(* Logix 5000 project; controller AMANA_DC_PLANT_01 vendor 1 type 14 code 164 rev 31.12; software revision 31.02; part 7 of 9 *)
(* tags used below, declared in another part *)
   Barcode_Longest : DINT;
   Barcode_Shortest : DINT;
   Comma : STRING;
   Counters : COUNTER[16];
   NULL_String : STRING;
   PRE_SET_COMMA_POSITION_1 : DINT;
   SCANNER_ClearPack_DATA : Keyence_2_Barcode;
   SCANNER_LN4_DATA : Keyence_2_Barcode;
   SCANNER_LN67MERGE_DATA : Keyence_2_Barcode;
   SCANNER_LN6_DATA : Keyence_2_Barcode;
   SCANNER_LN7_DATA : Keyence_2_Barcode;
   Read_From_Clearpack : INT[16];
(* OH_BARCODE_SCAN, continued *)

ROUTINE R01_CLEARPACK   (* ladder *)
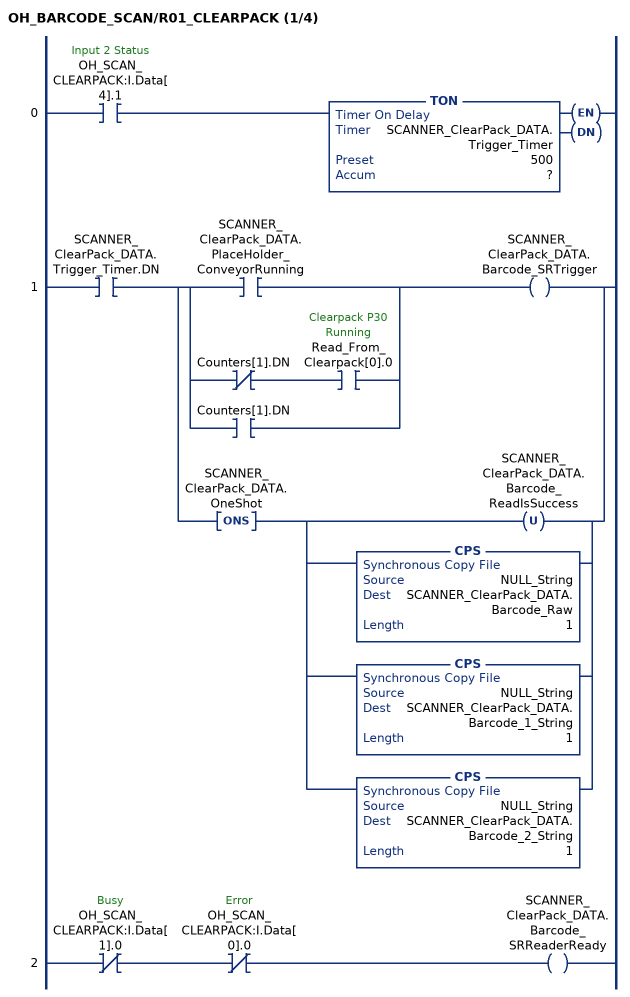
   0: XIC(OH_SCAN_CLEARPACK:I.Data[4].1)TON(SCANNER_ClearPack_DATA.Trigger_Timer,?,?);
   1: XIC(SCANNER_ClearPack_DATA.Trigger_Timer.DN)[[XIC(SCANNER_ClearPack_DATA.PlaceHolder_ConveyorRunning) ,XIO(Counters[1].DN) XIC(Read_From_Clearpack[0].0) ,XIC(Counters[1].DN) ] OTE(SCANNER_ClearPack_DATA.Barcode_SRTrigger) ,ONS(SCANNER_ClearPack_DATA.OneShot) [OTU(SCANNER_ClearPack_DATA.Barcode_ReadIsSuccess) ,CPS(NULL_String,SCANNER_ClearPack_DATA.Barcode_Raw,1) ,CPS(NULL_String,SCANNER_ClearPack_DATA.Barcode_1_String,1) ,CPS(NULL_String,SCANNER_ClearPack_DATA.Barcode_2_String,1) ] ];
   2: XIO(OH_SCAN_CLEARPACK:I.Data[1].0)XIO(OH_SCAN_CLEARPACK:I.Data[0].0)OTE(SCANNER_ClearPack_DATA.Barcode_SRReaderReady);
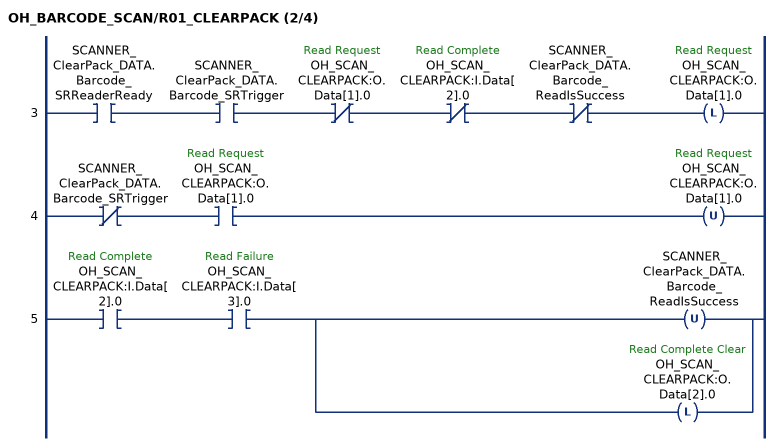
   3: XIC(SCANNER_ClearPack_DATA.Barcode_SRReaderReady)XIC(SCANNER_ClearPack_DATA.Barcode_SRTrigger)XIO(OH_SCAN_CLEARPACK:O.Data[1].0)XIO(OH_SCAN_CLEARPACK:I.Data[2].0)XIO(SCANNER_ClearPack_DATA.Barcode_ReadIsSuccess)OTL(OH_SCAN_CLEARPACK:O.Data[1].0);
   4: XIO(SCANNER_ClearPack_DATA.Barcode_SRTrigger)XIC(OH_SCAN_CLEARPACK:O.Data[1].0)OTU(OH_SCAN_CLEARPACK:O.Data[1].0);
   5: XIC(OH_SCAN_CLEARPACK:I.Data[2].0)XIC(OH_SCAN_CLEARPACK:I.Data[3].0)[OTU(SCANNER_ClearPack_DATA.Barcode_ReadIsSuccess) ,OTL(OH_SCAN_CLEARPACK:O.Data[2].0) ];
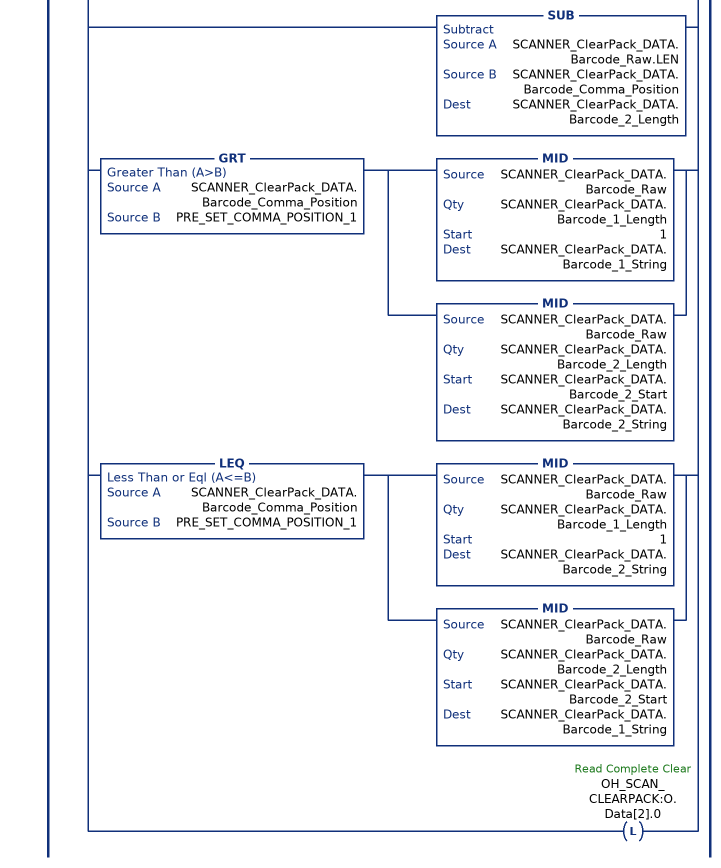
   6: XIC(OH_SCAN_CLEARPACK:I.Data[2].0)XIO(OH_SCAN_CLEARPACK:I.Data[3].0)LIM(Barcode_Shortest,OH_SCAN_CLEARPACK:I.Data[42],Barcode_Longest)[OTL(SCANNER_ClearPack_DATA.Barcode_ReadIsSuccess) ,SUB(OH_SCAN_CLEARPACK:I.Data[42],1,SCANNER_ClearPack_DATA.Barcode_Raw.LEN) ,CPS(OH_SCAN_CLEARPACK:I.Data[44],SCANNER_ClearPack_DATA.Barcode_Raw.DATA[0],SCANNER_ClearPack_DATA.Barcode_Raw.LEN) ,FIND(SCANNER_ClearPack_DATA.Barcode_Raw,Comma,1,SCANNER_ClearPack_DATA.Barcode_Comma_Position) ,SUB(SCANNER_ClearPack_DATA.Barcode_Comma_Position,1,SCANNER_ClearPack_DATA.Barcode_1_Length) ,ADD(SCANNER_ClearPack_DATA.Barcode_Comma_Position,1,SCANNER_ClearPack_DATA.Barcode_2_Start) ,SUB(SCANNER_ClearPack_DATA.Barcode_Raw.LEN,SCANNER_ClearPack_DATA.Barcode_Comma_Position,SCANNER_ClearPack_DATA.Barcode_2_Length) ,GRT(SCANNER_ClearPack_DATA.Barcode_Comma_Position,PRE_SET_COMMA_POSITION_1) [MID(SCANNER_ClearPack_DATA.Barcode_Raw,SCANNER_ClearPack_DATA.Barcode_1_Length,1,SCANNER_ClearPack_DATA.Barcode_1_String) ,MID(SCANNER_ClearPack_DATA.Barcode_Raw,SCANNER_ClearPack_DATA.Barcode_2_Length,SCANNER_ClearPack_DATA.Barcode_2_Start,SCANNER_ClearPack_DATA.Barcode_2_String) ] ,LEQ(SCANNER_ClearPack_DATA.Barcode_Comma_Position,PRE_SET_COMMA_POSITION_1) [MID(SCANNER_ClearPack_DATA.Barcode_Raw,SCANNER_ClearPack_DATA.Barcode_1_Length,1,SCANNER_ClearPack_DATA.Barcode_2_String) ,MID(SCANNER_ClearPack_DATA.Barcode_Raw,SCANNER_ClearPack_DATA.Barcode_2_Length,SCANNER_ClearPack_DATA.Barcode_2_Start,SCANNER_ClearPack_DATA.Barcode_1_String) ] ,OTL(OH_SCAN_CLEARPACK:O.Data[2].0) ];
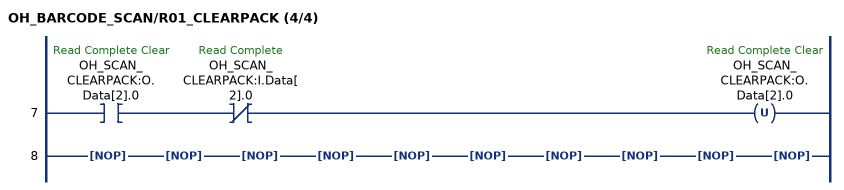
   7: XIC(OH_SCAN_CLEARPACK:O.Data[2].0)XIO(OH_SCAN_CLEARPACK:I.Data[2].0)OTU(OH_SCAN_CLEARPACK:O.Data[2].0);
   8: NOP()NOP()NOP()NOP()NOP()NOP()NOP()NOP()NOP()NOP();
END_ROUTINE

ROUTINE R02_LN4   (* ladder *)
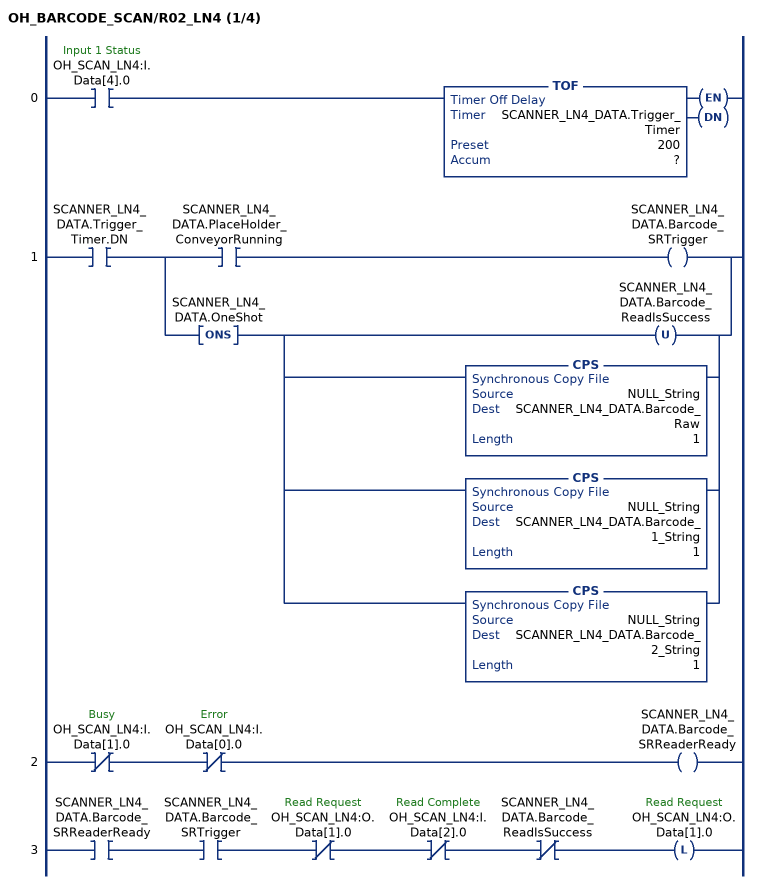
   0: XIC(OH_SCAN_LN4:I.Data[4].0)TOF(SCANNER_LN4_DATA.Trigger_Timer,?,?);
   1: XIC(SCANNER_LN4_DATA.Trigger_Timer.DN)[XIC(SCANNER_LN4_DATA.PlaceHolder_ConveyorRunning) OTE(SCANNER_LN4_DATA.Barcode_SRTrigger) ,ONS(SCANNER_LN4_DATA.OneShot) [OTU(SCANNER_LN4_DATA.Barcode_ReadIsSuccess) ,CPS(NULL_String,SCANNER_LN4_DATA.Barcode_Raw,1) ,CPS(NULL_String,SCANNER_LN4_DATA.Barcode_1_String,1) ,CPS(NULL_String,SCANNER_LN4_DATA.Barcode_2_String,1) ] ];
   2: XIO(OH_SCAN_LN4:I.Data[1].0)XIO(OH_SCAN_LN4:I.Data[0].0)OTE(SCANNER_LN4_DATA.Barcode_SRReaderReady);
   3: XIC(SCANNER_LN4_DATA.Barcode_SRReaderReady)XIC(SCANNER_LN4_DATA.Barcode_SRTrigger)XIO(OH_SCAN_LN4:O.Data[1].0)XIO(OH_SCAN_LN4:I.Data[2].0)XIO(SCANNER_LN4_DATA.Barcode_ReadIsSuccess)OTL(OH_SCAN_LN4:O.Data[1].0);
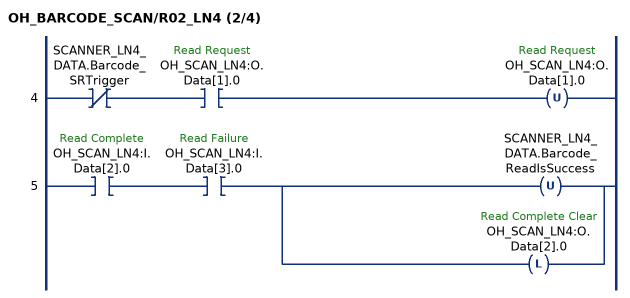
   4: XIO(SCANNER_LN4_DATA.Barcode_SRTrigger)XIC(OH_SCAN_LN4:O.Data[1].0)OTU(OH_SCAN_LN4:O.Data[1].0);
   5: XIC(OH_SCAN_LN4:I.Data[2].0)XIC(OH_SCAN_LN4:I.Data[3].0)[OTU(SCANNER_LN4_DATA.Barcode_ReadIsSuccess) ,OTL(OH_SCAN_LN4:O.Data[2].0) ];
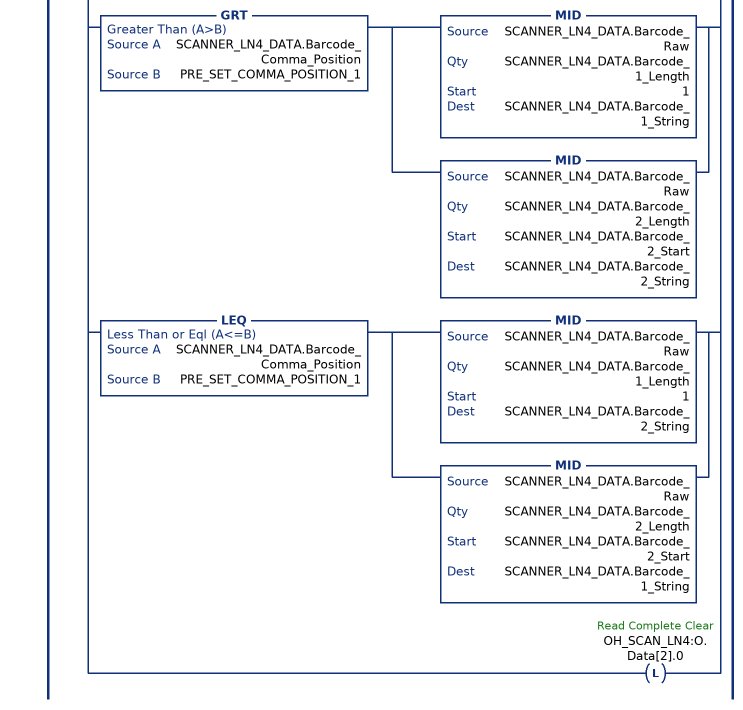
   6: XIC(OH_SCAN_LN4:I.Data[2].0)XIO(OH_SCAN_LN4:I.Data[3].0)LIM(Barcode_Shortest,OH_SCAN_LN4:I.Data[42],Barcode_Longest)[OTL(SCANNER_LN4_DATA.Barcode_ReadIsSuccess) ,SUB(OH_SCAN_LN4:I.Data[42],1,SCANNER_LN4_DATA.Barcode_Raw.LEN) ,CPS(OH_SCAN_LN4:I.Data[44],SCANNER_LN4_DATA.Barcode_Raw.DATA[0],SCANNER_LN4_DATA.Barcode_Raw.LEN) ,FIND(SCANNER_LN4_DATA.Barcode_Raw,Comma,1,SCANNER_LN4_DATA.Barcode_Comma_Position) ,SUB(SCANNER_LN4_DATA.Barcode_Comma_Position,1,SCANNER_LN4_DATA.Barcode_1_Length) ,ADD(SCANNER_LN4_DATA.Barcode_Comma_Position,1,SCANNER_LN4_DATA.Barcode_2_Start) ,SUB(SCANNER_LN4_DATA.Barcode_Raw.LEN,SCANNER_LN4_DATA.Barcode_Comma_Position,SCANNER_LN4_DATA.Barcode_2_Length) ,GRT(SCANNER_LN4_DATA.Barcode_Comma_Position,PRE_SET_COMMA_POSITION_1) [MID(SCANNER_LN4_DATA.Barcode_Raw,SCANNER_LN4_DATA.Barcode_1_Length,1,SCANNER_LN4_DATA.Barcode_1_String) ,MID(SCANNER_LN4_DATA.Barcode_Raw,SCANNER_LN4_DATA.Barcode_2_Length,SCANNER_LN4_DATA.Barcode_2_Start,SCANNER_LN4_DATA.Barcode_2_String) ] ,LEQ(SCANNER_LN4_DATA.Barcode_Comma_Position,PRE_SET_COMMA_POSITION_1) [MID(SCANNER_LN4_DATA.Barcode_Raw,SCANNER_LN4_DATA.Barcode_1_Length,1,SCANNER_LN4_DATA.Barcode_2_String) ,MID(SCANNER_LN4_DATA.Barcode_Raw,SCANNER_LN4_DATA.Barcode_2_Length,SCANNER_LN4_DATA.Barcode_2_Start,SCANNER_LN4_DATA.Barcode_1_String) ] ,OTL(OH_SCAN_LN4:O.Data[2].0) ];
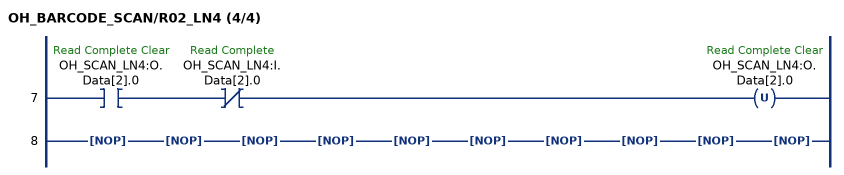
   7: XIC(OH_SCAN_LN4:O.Data[2].0)XIO(OH_SCAN_LN4:I.Data[2].0)OTU(OH_SCAN_LN4:O.Data[2].0);
   8: NOP()NOP()NOP()NOP()NOP()NOP()NOP()NOP()NOP()NOP();
END_ROUTINE

ROUTINE R03_LN6   (* ladder *)
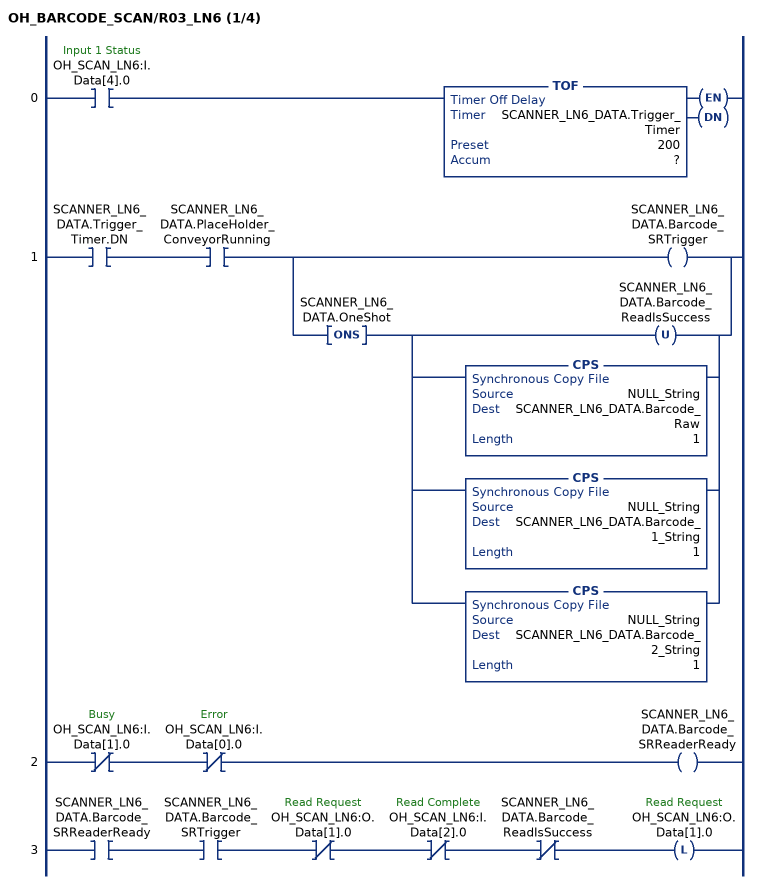
   0: XIC(OH_SCAN_LN6:I.Data[4].0)TOF(SCANNER_LN6_DATA.Trigger_Timer,?,?);
   1: XIC(SCANNER_LN6_DATA.Trigger_Timer.DN)XIC(SCANNER_LN6_DATA.PlaceHolder_ConveyorRunning)[OTE(SCANNER_LN6_DATA.Barcode_SRTrigger) ,ONS(SCANNER_LN6_DATA.OneShot) [OTU(SCANNER_LN6_DATA.Barcode_ReadIsSuccess) ,CPS(NULL_String,SCANNER_LN6_DATA.Barcode_Raw,1) ,CPS(NULL_String,SCANNER_LN6_DATA.Barcode_1_String,1) ,CPS(NULL_String,SCANNER_LN6_DATA.Barcode_2_String,1) ] ];
   2: XIO(OH_SCAN_LN6:I.Data[1].0)XIO(OH_SCAN_LN6:I.Data[0].0)OTE(SCANNER_LN6_DATA.Barcode_SRReaderReady);
   3: XIC(SCANNER_LN6_DATA.Barcode_SRReaderReady)XIC(SCANNER_LN6_DATA.Barcode_SRTrigger)XIO(OH_SCAN_LN6:O.Data[1].0)XIO(OH_SCAN_LN6:I.Data[2].0)XIO(SCANNER_LN6_DATA.Barcode_ReadIsSuccess)OTL(OH_SCAN_LN6:O.Data[1].0);
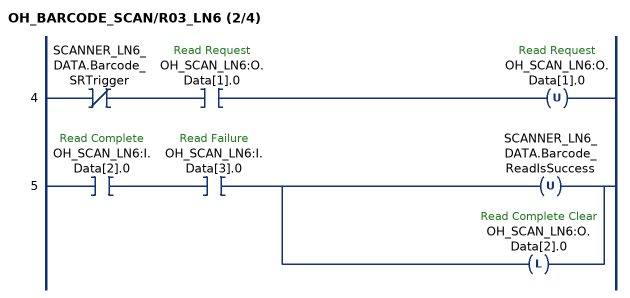
   4: XIO(SCANNER_LN6_DATA.Barcode_SRTrigger)XIC(OH_SCAN_LN6:O.Data[1].0)OTU(OH_SCAN_LN6:O.Data[1].0);
   5: XIC(OH_SCAN_LN6:I.Data[2].0)XIC(OH_SCAN_LN6:I.Data[3].0)[OTU(SCANNER_LN6_DATA.Barcode_ReadIsSuccess) ,OTL(OH_SCAN_LN6:O.Data[2].0) ];
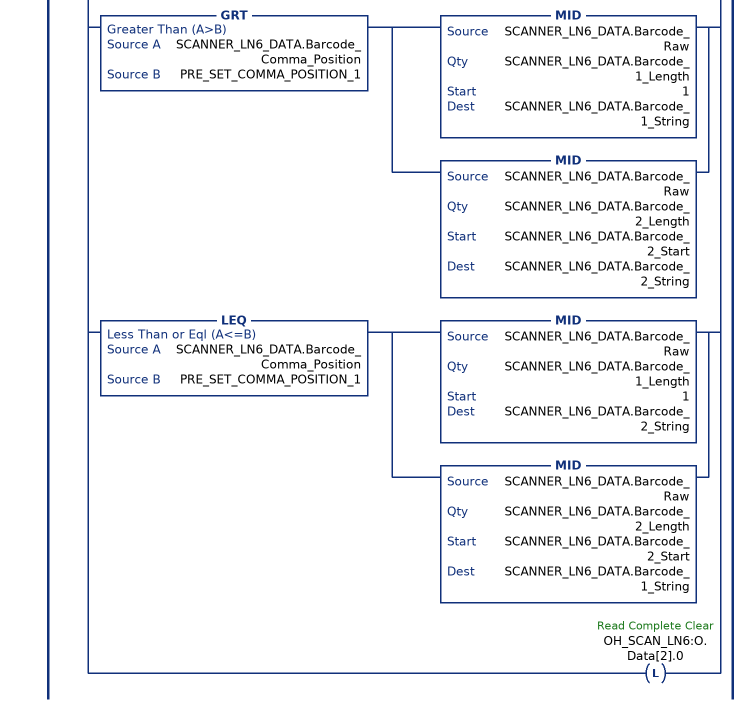
   6: XIC(OH_SCAN_LN6:I.Data[2].0)XIO(OH_SCAN_LN6:I.Data[3].0)LIM(Barcode_Shortest,OH_SCAN_LN6:I.Data[42],Barcode_Longest)[OTL(SCANNER_LN6_DATA.Barcode_ReadIsSuccess) ,SUB(OH_SCAN_LN6:I.Data[42],1,SCANNER_LN6_DATA.Barcode_Raw.LEN) ,CPS(OH_SCAN_LN6:I.Data[44],SCANNER_LN6_DATA.Barcode_Raw.DATA[0],SCANNER_LN6_DATA.Barcode_Raw.LEN) ,FIND(SCANNER_LN6_DATA.Barcode_Raw,Comma,1,SCANNER_LN6_DATA.Barcode_Comma_Position) ,SUB(SCANNER_LN6_DATA.Barcode_Comma_Position,1,SCANNER_LN6_DATA.Barcode_1_Length) ,ADD(SCANNER_LN6_DATA.Barcode_Comma_Position,1,SCANNER_LN6_DATA.Barcode_2_Start) ,SUB(SCANNER_LN6_DATA.Barcode_Raw.LEN,SCANNER_LN6_DATA.Barcode_Comma_Position,SCANNER_LN6_DATA.Barcode_2_Length) ,GRT(SCANNER_LN6_DATA.Barcode_Comma_Position,PRE_SET_COMMA_POSITION_1) [MID(SCANNER_LN6_DATA.Barcode_Raw,SCANNER_LN6_DATA.Barcode_1_Length,1,SCANNER_LN6_DATA.Barcode_1_String) ,MID(SCANNER_LN6_DATA.Barcode_Raw,SCANNER_LN6_DATA.Barcode_2_Length,SCANNER_LN6_DATA.Barcode_2_Start,SCANNER_LN6_DATA.Barcode_2_String) ] ,LEQ(SCANNER_LN6_DATA.Barcode_Comma_Position,PRE_SET_COMMA_POSITION_1) [MID(SCANNER_LN6_DATA.Barcode_Raw,SCANNER_LN6_DATA.Barcode_1_Length,1,SCANNER_LN6_DATA.Barcode_2_String) ,MID(SCANNER_LN6_DATA.Barcode_Raw,SCANNER_LN6_DATA.Barcode_2_Length,SCANNER_LN6_DATA.Barcode_2_Start,SCANNER_LN6_DATA.Barcode_1_String) ] ,OTL(OH_SCAN_LN6:O.Data[2].0) ];
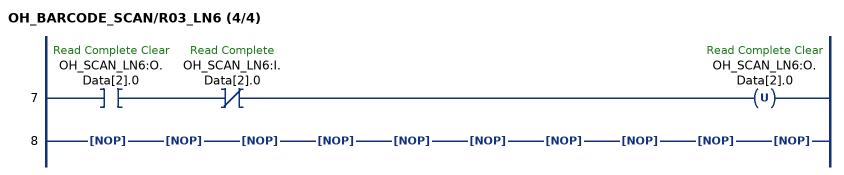
   7: XIC(OH_SCAN_LN6:O.Data[2].0)XIO(OH_SCAN_LN6:I.Data[2].0)OTU(OH_SCAN_LN6:O.Data[2].0);
   8: NOP()NOP()NOP()NOP()NOP()NOP()NOP()NOP()NOP()NOP();
END_ROUTINE

ROUTINE R04_LN7   (* ladder *)
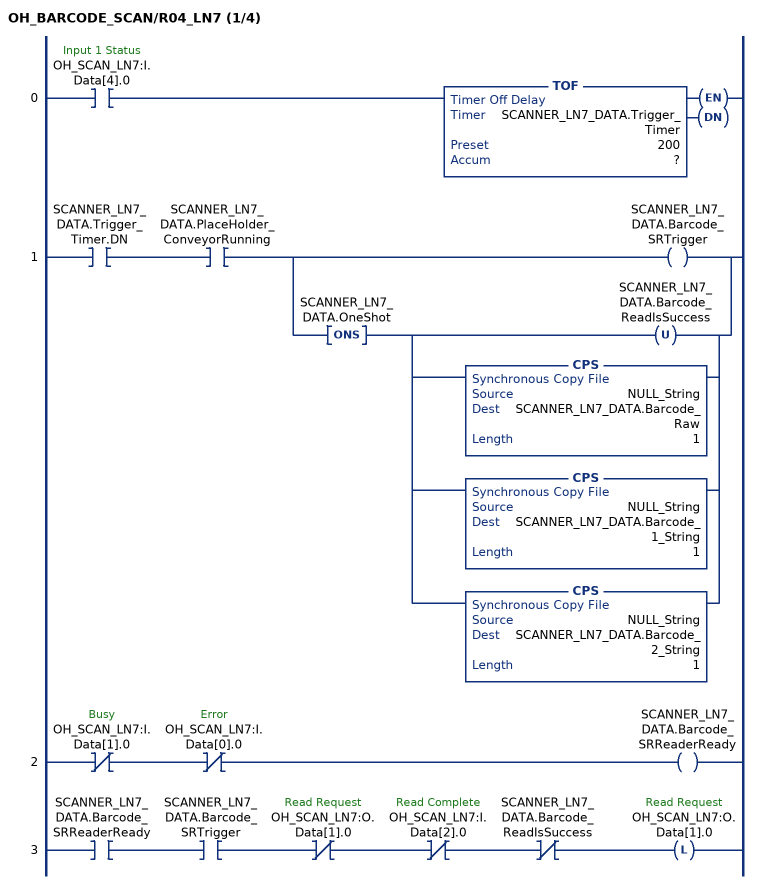
   0: XIC(OH_SCAN_LN7:I.Data[4].0)TOF(SCANNER_LN7_DATA.Trigger_Timer,?,?);
   1: XIC(SCANNER_LN7_DATA.Trigger_Timer.DN)XIC(SCANNER_LN7_DATA.PlaceHolder_ConveyorRunning)[OTE(SCANNER_LN7_DATA.Barcode_SRTrigger) ,ONS(SCANNER_LN7_DATA.OneShot) [OTU(SCANNER_LN7_DATA.Barcode_ReadIsSuccess) ,CPS(NULL_String,SCANNER_LN7_DATA.Barcode_Raw,1) ,CPS(NULL_String,SCANNER_LN7_DATA.Barcode_1_String,1) ,CPS(NULL_String,SCANNER_LN7_DATA.Barcode_2_String,1) ] ];
   2: XIO(OH_SCAN_LN7:I.Data[1].0)XIO(OH_SCAN_LN7:I.Data[0].0)OTE(SCANNER_LN7_DATA.Barcode_SRReaderReady);
   3: XIC(SCANNER_LN7_DATA.Barcode_SRReaderReady)XIC(SCANNER_LN7_DATA.Barcode_SRTrigger)XIO(OH_SCAN_LN7:O.Data[1].0)XIO(OH_SCAN_LN7:I.Data[2].0)XIO(SCANNER_LN7_DATA.Barcode_ReadIsSuccess)OTL(OH_SCAN_LN7:O.Data[1].0);
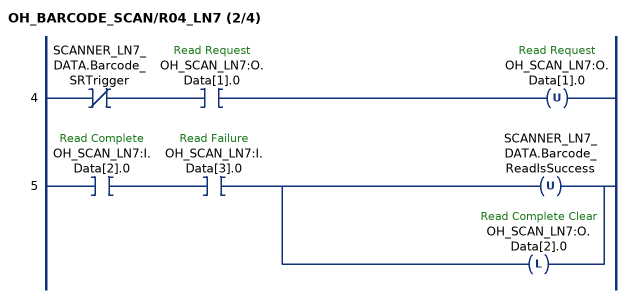
   4: XIO(SCANNER_LN7_DATA.Barcode_SRTrigger)XIC(OH_SCAN_LN7:O.Data[1].0)OTU(OH_SCAN_LN7:O.Data[1].0);
   5: XIC(OH_SCAN_LN7:I.Data[2].0)XIC(OH_SCAN_LN7:I.Data[3].0)[OTU(SCANNER_LN7_DATA.Barcode_ReadIsSuccess) ,OTL(OH_SCAN_LN7:O.Data[2].0) ];
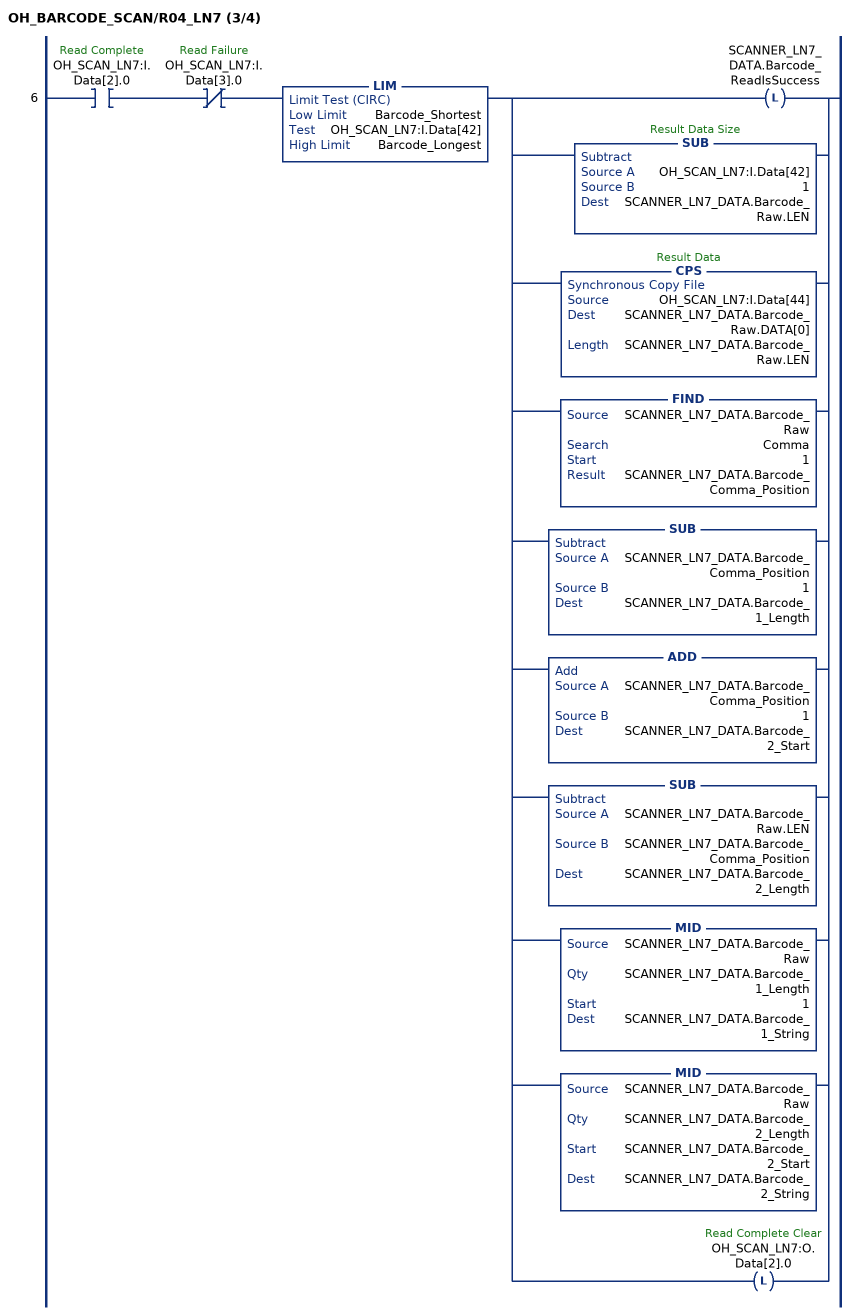
   6: XIC(OH_SCAN_LN7:I.Data[2].0)XIO(OH_SCAN_LN7:I.Data[3].0)LIM(Barcode_Shortest,OH_SCAN_LN7:I.Data[42],Barcode_Longest)[OTL(SCANNER_LN7_DATA.Barcode_ReadIsSuccess) ,SUB(OH_SCAN_LN7:I.Data[42],1,SCANNER_LN7_DATA.Barcode_Raw.LEN) ,CPS(OH_SCAN_LN7:I.Data[44],SCANNER_LN7_DATA.Barcode_Raw.DATA[0],SCANNER_LN7_DATA.Barcode_Raw.LEN) ,FIND(SCANNER_LN7_DATA.Barcode_Raw,Comma,1,SCANNER_LN7_DATA.Barcode_Comma_Position) ,SUB(SCANNER_LN7_DATA.Barcode_Comma_Position,1,SCANNER_LN7_DATA.Barcode_1_Length) ,ADD(SCANNER_LN7_DATA.Barcode_Comma_Position,1,SCANNER_LN7_DATA.Barcode_2_Start) ,SUB(SCANNER_LN7_DATA.Barcode_Raw.LEN,SCANNER_LN7_DATA.Barcode_Comma_Position,SCANNER_LN7_DATA.Barcode_2_Length) ,MID(SCANNER_LN7_DATA.Barcode_Raw,SCANNER_LN7_DATA.Barcode_1_Length,1,SCANNER_LN7_DATA.Barcode_1_String) ,MID(SCANNER_LN7_DATA.Barcode_Raw,SCANNER_LN7_DATA.Barcode_2_Length,SCANNER_LN7_DATA.Barcode_2_Start,SCANNER_LN7_DATA.Barcode_2_String) ,OTL(OH_SCAN_LN7:O.Data[2].0) ];
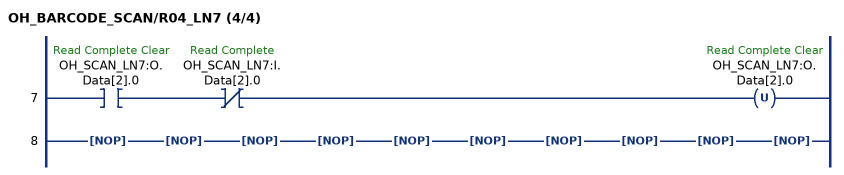
   7: XIC(OH_SCAN_LN7:O.Data[2].0)XIO(OH_SCAN_LN7:I.Data[2].0)OTU(OH_SCAN_LN7:O.Data[2].0);
   8: NOP()NOP()NOP()NOP()NOP()NOP()NOP()NOP()NOP()NOP();
END_ROUTINE

ROUTINE R05_LN67MERGE   (* ladder *)
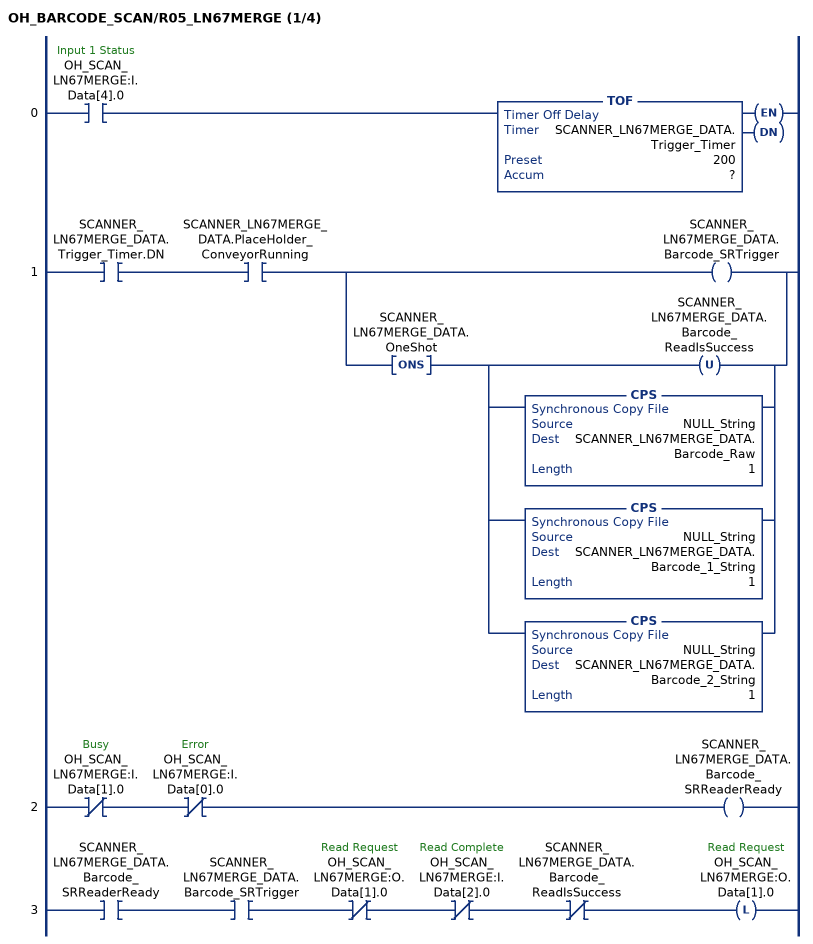
   0: XIC(OH_SCAN_LN67MERGE:I.Data[4].0)TOF(SCANNER_LN67MERGE_DATA.Trigger_Timer,?,?);
   1: XIC(SCANNER_LN67MERGE_DATA.Trigger_Timer.DN)XIC(SCANNER_LN67MERGE_DATA.PlaceHolder_ConveyorRunning)[OTE(SCANNER_LN67MERGE_DATA.Barcode_SRTrigger) ,ONS(SCANNER_LN67MERGE_DATA.OneShot) [OTU(SCANNER_LN67MERGE_DATA.Barcode_ReadIsSuccess) ,CPS(NULL_String,SCANNER_LN67MERGE_DATA.Barcode_Raw,1) ,CPS(NULL_String,SCANNER_LN67MERGE_DATA.Barcode_1_String,1) ,CPS(NULL_String,SCANNER_LN67MERGE_DATA.Barcode_2_String,1) ] ];
   2: XIO(OH_SCAN_LN67MERGE:I.Data[1].0)XIO(OH_SCAN_LN67MERGE:I.Data[0].0)OTE(SCANNER_LN67MERGE_DATA.Barcode_SRReaderReady);
   3: XIC(SCANNER_LN67MERGE_DATA.Barcode_SRReaderReady)XIC(SCANNER_LN67MERGE_DATA.Barcode_SRTrigger)XIO(OH_SCAN_LN67MERGE:O.Data[1].0)XIO(OH_SCAN_LN67MERGE:I.Data[2].0)XIO(SCANNER_LN67MERGE_DATA.Barcode_ReadIsSuccess)OTL(OH_SCAN_LN67MERGE:O.Data[1].0);
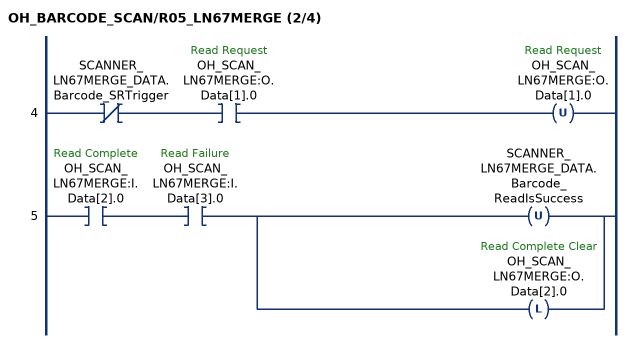
   4: XIO(SCANNER_LN67MERGE_DATA.Barcode_SRTrigger)XIC(OH_SCAN_LN67MERGE:O.Data[1].0)OTU(OH_SCAN_LN67MERGE:O.Data[1].0);
   5: XIC(OH_SCAN_LN67MERGE:I.Data[2].0)XIC(OH_SCAN_LN67MERGE:I.Data[3].0)[OTU(SCANNER_LN67MERGE_DATA.Barcode_ReadIsSuccess) ,OTL(OH_SCAN_LN67MERGE:O.Data[2].0) ];
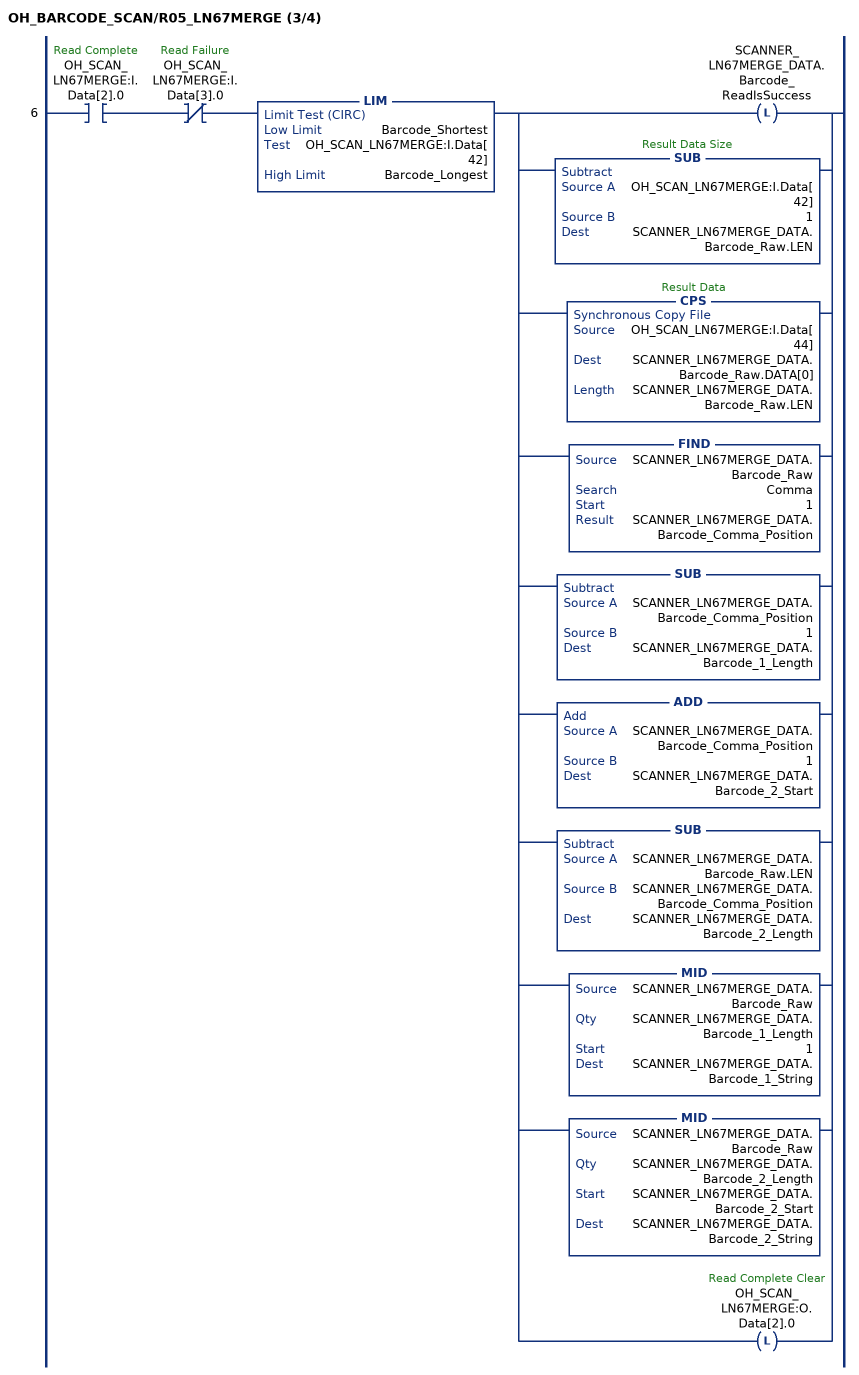
   6: XIC(OH_SCAN_LN67MERGE:I.Data[2].0)XIO(OH_SCAN_LN67MERGE:I.Data[3].0)LIM(Barcode_Shortest,OH_SCAN_LN67MERGE:I.Data[42],Barcode_Longest)[OTL(SCANNER_LN67MERGE_DATA.Barcode_ReadIsSuccess) ,SUB(OH_SCAN_LN67MERGE:I.Data[42],1,SCANNER_LN67MERGE_DATA.Barcode_Raw.LEN) ,CPS(OH_SCAN_LN67MERGE:I.Data[44],SCANNER_LN67MERGE_DATA.Barcode_Raw.DATA[0],SCANNER_LN67MERGE_DATA.Barcode_Raw.LEN) ,FIND(SCANNER_LN67MERGE_DATA.Barcode_Raw,Comma,1,SCANNER_LN67MERGE_DATA.Barcode_Comma_Position) ,SUB(SCANNER_LN67MERGE_DATA.Barcode_Comma_Position,1,SCANNER_LN67MERGE_DATA.Barcode_1_Length) ,ADD(SCANNER_LN67MERGE_DATA.Barcode_Comma_Position,1,SCANNER_LN67MERGE_DATA.Barcode_2_Start) ,SUB(SCANNER_LN67MERGE_DATA.Barcode_Raw.LEN,SCANNER_LN67MERGE_DATA.Barcode_Comma_Position,SCANNER_LN67MERGE_DATA.Barcode_2_Length) ,MID(SCANNER_LN67MERGE_DATA.Barcode_Raw,SCANNER_LN67MERGE_DATA.Barcode_1_Length,1,SCANNER_LN67MERGE_DATA.Barcode_1_String) ,MID(SCANNER_LN67MERGE_DATA.Barcode_Raw,SCANNER_LN67MERGE_DATA.Barcode_2_Length,SCANNER_LN67MERGE_DATA.Barcode_2_Start,SCANNER_LN67MERGE_DATA.Barcode_2_String) ,OTL(OH_SCAN_LN67MERGE:O.Data[2].0) ];
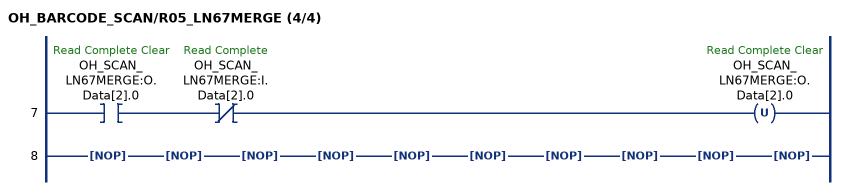
   7: XIC(OH_SCAN_LN67MERGE:O.Data[2].0)XIO(OH_SCAN_LN67MERGE:I.Data[2].0)OTU(OH_SCAN_LN67MERGE:O.Data[2].0);
   8: NOP()NOP()NOP()NOP()NOP()NOP()NOP()NOP()NOP()NOP();
END_ROUTINE
